INTERFACE I_Cylinder

PROPERTY PUBLIC Config : REFERENCE TO ST_CylinderConfig
GET
END_GET
END_PROPERTY

PROPERTY PUBLIC inHP : BOOL
GET
END_GET
END_PROPERTY

PROPERTY PUBLIC interlockHP : BOOL
GET
END_GET
SET
END_SET
END_PROPERTY

PROPERTY PUBLIC interlockWP : BOOL
GET
END_GET
SET
END_SET
END_PROPERTY

PROPERTY PUBLIC inWP : BOOL
GET
END_GET
END_PROPERTY

METHOD PUBLIC moveToHP
VAR_INPUT
	Response		: REFERENCE TO TcNexa_Components_TcProcess.FB_MethodResponse;
END_VAR
END_METHOD

METHOD PUBLIC moveToWP
VAR_INPUT
	Response		: REFERENCE TO TcNexa_Components_TcProcess.FB_MethodResponse;
END_VAR
END_METHOD

METHOD PUBLIC off
VAR_INPUT
END_VAR
END_METHOD

END_INTERFACE

(* stored: Version 1.1.0.1, ProductVersion 3.1.4024.12
   Itf I_Cylinder: Id {c5f5e301-2dad-4980-9099-2aea1dcf63b3}
   Property Config: Id {1a8f4113-562f-4303-a4ac-e3dc7a6f21e2}
   Get Get: Id {9505e93f-1af3-46af-86ae-30758fa99b8a}
   Property inHP: Id {39c2d449-199d-46ee-910a-ba1ff3cc2305}
   Get Get: Id {f6860966-e6c9-4f2d-a24c-d7a7d19957d1}
   Property interlockHP: Id {43421e2d-0c30-06d1-0797-074421230813}
   Get Get: Id {ba540fc3-33c1-087d-3147-014199a12d3d}
   Set Set: Id {798686c5-ae5d-0db3-36b6-f8457c3b0779}
   Property interlockWP: Id {efa5008d-2cad-0334-0f11-566d2c6c8df0}
   Get Get: Id {edfa9e16-cb25-0d13-1ab2-72eee85ebb7f}
   Set Set: Id {c10ae8a7-f5c9-0a38-3ae5-b82b9eba5eed}
   Property inWP: Id {3c1cb09a-ef9f-4672-9198-506b4f224e44}
   Get Get: Id {1ce88175-8a16-471c-9864-81c4b17a7be0}
   Method moveToHP: Id {9d2a05ac-b15a-4400-a8bf-7b7682136c31}
   Method moveToWP: Id {4f67f11d-8dac-44c5-b1ee-185be19b9b38}
   Method off: Id {87d49e7f-c993-4cae-975b-02234bb3e223} *)
